Fanuc KAREL source: kb00128.KL

-- PROVISIONAL review KL for V940-1; original PC SHA256 664ee398ae5e9e45a904fb4f01307974fbd4f49f0cf21966537aa03abb745968
-- Incomplete behavior may be omitted. Consult companion uncertainty JSON. Do not deploy.
PROGRAM KB00128
%NOLOCKGROUP
BEGIN
  -- V9_ZERO_TABLE_METADATA_HINT layout=0002_ascii; no indexed target words; source/name/runtime held
  -- UNRESOLVED_PC offsets 5-28; opcodes 27,22,1C,31,4A
  -- UNRESOLVED_PC offsets 33-37; opcodes 7F
END KB00128
